// TIA Portal V18 export
DATA_BLOCK "Metering Program Parameters"   // DB45
{ S7_Optimized_Access := 'FALSE' }
VERSION : 0.1
// stored: AutoNumber true, DBAccessibleFromOPCUA true, IsOnlyStoredInLoadMemory false, IsWriteProtectedInAS false
   VAR RETAIN
      "program No site" : Int;
      "Program No screen" : Int;
      "Receipe Program No" : DInt;
      "Receipe Set Flowrate" : Real;
      "Receipe Set qty" : Real;
      "Receipe Description" : String[12];
      "Receipe Flowrate Adjustment A" : Real;
      "Receipe Flowrate Adjustment B" : Real;
      "Current Program" : Struct
         "Set Flowrate" : Real;
         "Set qty" : Real;
         Description : String[12];
         "Flowrate Adjustment A" : Real;
         "Flowrate Adjustment B" : Real;
         "Set Flowrate snuffback" : Real;
         "Set qty snuffback" : Real;
         "Set delay snuffback" : Time;
      END_STRUCT;
      "Current program No" : DInt;
      "Min Mixed Flowrate Ml" : Real;
      "Max Mixed Flowrate Ml" : Real;
      "Max A Flowrate Ml" : Real;
      "Max B Flowrate Ml" : Real;
      "Receipe Set Flowrate snuffback" : Real;
      "Receipe Set Qty snuffback" : Real;
      "Receipe Set delay snuffback" : Time;
   END_VAR
BEGIN
END_DATA_BLOCK
